{attribute 'qualified_only'}
//{attribute 'strict'}
TYPE SectionStatus :
(
	IDLE,
	ALIGNING,
	ACTIVE,
	CLEARING,
	COMPLETE,
	
	size
);
END_TYPE

(* stored: Version 1.1.0.1, ProductVersion 3.1.4024.11
   DUT SectionStatus: Id {9750fdd6-c9e6-4c18-b005-35290999abad} *)
